{attribute 'qualified_only'}
{attribute 'to_string'}
//All of the CAN IDs and what they correspond to

TYPE Drive_error_mapping :
(
	none := -1,
	Motor_overload := 0,
	Heatsink_overtemp := 1,
	Motor_overtemp := 2,
	Drive_overtemp := 3,
	Control_voltage := 4,
	Feedback := 5,
	Commutation := 6,
	Overcurrent := 7,
	Overvoltage := 8,
	Undervoltage := 9,
	Supply_phase := 10,
	Psn_dev := 11,
	Comms := 12,
	Overtravel := 13
	
	
)INT := none;
END_TYPE

(* stored: Version 1.1.0.1
   DUT Drive_error_mapping: Id {9ee6572c-5032-46c2-b837-de7ffdd79493} *)
